FUNCTION_BLOCK TcaRackFeeder EXTENDS TcoCore.TcoComponent

VAR_INPUT
	ref : REFERENCE TO TcaRackFeederRef;
END_VAR

VAR
	_status : TcaRackFeederStatus;
	_config : TcaRackFeederConfig;
	_service : TcaRackFeederService;
END_VAR

PROPERTY Config : REFERENCE TO TcaRackFeederConfig
GET
Config Ref= _config;
END_GET
SET
_config := Config;
END_SET
END_PROPERTY

{warning 'Methodenimplementierung hinzufügen'}
METHOD Restore : TcoCore.ITcoRestorable
END_METHOD

{warning 'Methodenimplementierung hinzufügen'}
(*~
	<docu>
		<summary>
		    Custom service (manual, maintenance) logic.
			This method must be implemented in derived class.
		</summary>			
	</docu>	
~*)
METHOD PROTECTED ServiceMode
END_METHOD

PROPERTY Status : REFERENCE TO TcaRackFeederStatus
GET
Status REF= _status;
END_GET
END_PROPERTY

END_FUNCTION_BLOCK

(* stored: Version 1.1.0.1
   POU TcaRackFeeder: Id {491823f4-bf55-40f2-9dc6-19dc420c158e}, SpecialFunc None
   Folder Functions: Id {a73bda7e-8f56-47cd-9168-de5eeaca9d2a}
   Folder Operations: Id {1e5d19b5-5904-4c05-b625-267e4ebbd52f}
   Folder States: Id {ef83b66c-6eb7-4a8e-9039-66ce8f0a6986}
   Folder Tasks: Id {e91973e5-a009-4993-a29b-89f80771f7bd}
   Property Config: Id {6c22c004-cb16-46db-8ade-11d87e25f356}
   Get Get: Id {169e9214-7036-41fd-bb75-2895b74d4f38}
   Set Set: Id {a53cf5ef-b155-44ab-90a1-87d93653f698}
   Method Restore: Id {a85fb066-a6cd-4a24-99b9-124aeeec9f21}
   Method ServiceMode: Id {551788e3-8e5a-4a29-a0a4-0a0bd04f6a1f}
   Property Status: Id {bdd2a1a1-45b9-4ddc-b040-b6a9716631da}
   Get Get: Id {320fb7fe-559d-4c79-ba78-5142752ba8ba} *)
